FUNCTION R2_ABS : REAL2
VAR_INPUT
	X : REAL2;
END_VAR


(*
version 1.1	10. mar. 2009
programmer 	hugo
tested by		tobias

R2_abs returns the absulute value of a double precision real.

*)

IF X.RX >= 0.0 THEN
	R2_ABS.RX := X.RX;
	R2_ABS.R1 := X.R1;
ELSE
	R2_ABS.RX := -X.RX;
	R2_ABS.R1 := -X.R1;
END_IF;


(* revision history
hm	21. mar. 2008	rev 1.0
	original version

hm	10. mar. 2009 rev 1.1
	real constants updated to new systax using dot

*)

END_FUNCTION

(* stored: Version 1.1.0.1, ProductVersion 3.1.4022.7
   POU R2_ABS: Id {3d5f686d-79ce-4980-b268-babb43996a8f}, SpecialFunc None *)
